TYPE ST_AxisParams :
STRUCT
	unit: STRING := 'mm';
	ref_vel: LREAL;
	max_vel: LREAL;
	max_acc: LREAL := 15000;
	max_dec: LREAL := 15000;
	def_acc: LREAL := 1500;
	def_dec: LREAL := 1500;
	def_jerk: LREAL := 2250;
	home_search: LREAL;
	home_sync: LREAL;
	man_fast: LREAL;
	man_slow: LREAL;
	dead_time: LREAL := 0.008;
	enc_scale: LREAL;
	enc_invert: BOOL;
	mot_invert: BOOL;
	max_current: UINT;
	holding_current: UINT := 100;
	voltage: UINT := 24000;
	resistance: UINT := 100;
	emf: UINT := 0;
	full_steps: UINT := 200;
	speed_range: USINT := 1;
	enc_supply: USINT := 50;
	enc_clock: USINT := 9;
	enc_multi_bits: USINT := 0;
	enc_single_bits: USINT := 32;
END_STRUCT
END_TYPE

(* stored: Version 1.1.0.1, ProductVersion 3.1.4020.12
   DUT ST_AxisParams: Id {3cafee99-db25-43c6-98e3-7fe336a53c10} *)
